{attribute 'GeneratedUsingTerminal: KL9528'}
{attribute addProperty BoxType "KL9528"}
{attribute addProperty Id "OverloadAT %I*BOOL0UndervoltageAT %I*BOOL0ResetAT %Q*BOOL0"}
{attribute addProperty CRC "2720558"}
{attribute addProperty Size "0"}
TYPE Channel_0029832E :
STRUCT
	{attribute addProperty Name "Overload"}
	Overload AT %I* : BOOL;
	{attribute addProperty Name "Undervoltage"}
	Undervoltage AT %I* : BOOL;
	{attribute addProperty Name "Reset"}
	Reset AT %Q* : BOOL;
END_STRUCT
END_TYPE

(* stored: Version 1.2.0.0, ProductVersion 3.1.4024.11
   DUT Channel_0029832E: Id {e329d4c1-2199-4aa4-aa8c-83116e973132} *)
